# EPICS autosave request: soft_iocs/meas_comp/iocBoot/iocmeas_comp_usb/auto_settings.req
file "USB1608G_settings.req", P=$(P1)
file "USB1608G_settings.req", P=$(P2)
file "USB1608G_2AO_settings.req", P=$(P3)
